FUNCTION PositionIsValid : BOOL
VAR_INPUT
	pair : REFERENCE TO PositionMaterials;
END_VAR

PositionIsValid := (
	pair.position <> -1 AND
	(
		pair.top <> '' OR
		pair.left <> '' OR
		pair.right <> '' OR
		pair.bottom <> '' OR
		
		pair.topLeft <> '' OR
		pair.topRight <> '' OR
		pair.bottomLeft <> '' OR
		pair.bottomRight <> ''
	));

END_FUNCTION

(* stored: Version 1.1.0.1, ProductVersion 3.1.4024.11
   POU PositionIsValid: Id {634a1648-c062-471b-b905-5d3fad291561}, SpecialFunc None *)
